PROGRAM Zuweisung
VAR

END_VAR

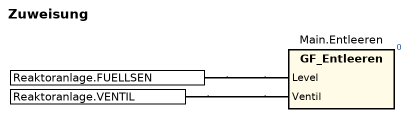
Main.Entleeren(Level := Reaktoranlage.FUELLSEN, Ventil := Reaktoranlage.VENTIL); // GF_Entleeren

END_PROGRAM

(* stored: Version 1.1.0.1, ProductVersion 3.1.4024.12
   POU Zuweisung: Id {6c34c34c-3732-41d0-aa22-455bcd3452a5}, SpecialFunc None *)
